# B&R Automation Studio project ACOPOStrakbyOk
Automation Studio 4.12.4.107 SP; technology packages: mappMotion 5.23.1

## Configuration Config1

CPU X20CP1586, AutomationRuntime E4.93, Build 4.1.2, Safety 0.0, Vc V4.72.6

### Task classes (Cpu.sw)
```
Cyclic#1 (cycle 800 us, tolerance 0 us):
  Vis <- Visualization.Vis.prg
Cyclic#4:
  StartMovem <- AssemblyControl.StartMovement.prg
DataObjects: McAcpSys
NcDataObjects: McDriveLog
Binaries: arsvcreg, udbdef, McAcpDrv, arflatprv, McProfGen, arcoal, FWRules, TCData, McAcpSim, ashwd, Config_1, ashwac, User, Config_4, sysconf, iomap, asfw, arconfig, Config_3, Config_2, Role
Libraries: McBase, McAxis, McAcpTrak, MpBase, operator, runtime, astime, AsIecCon, MpAxis, McAcpAx, AsBrStr, powerlnk, fileio, asepl, sys_lib
```

### Hardware
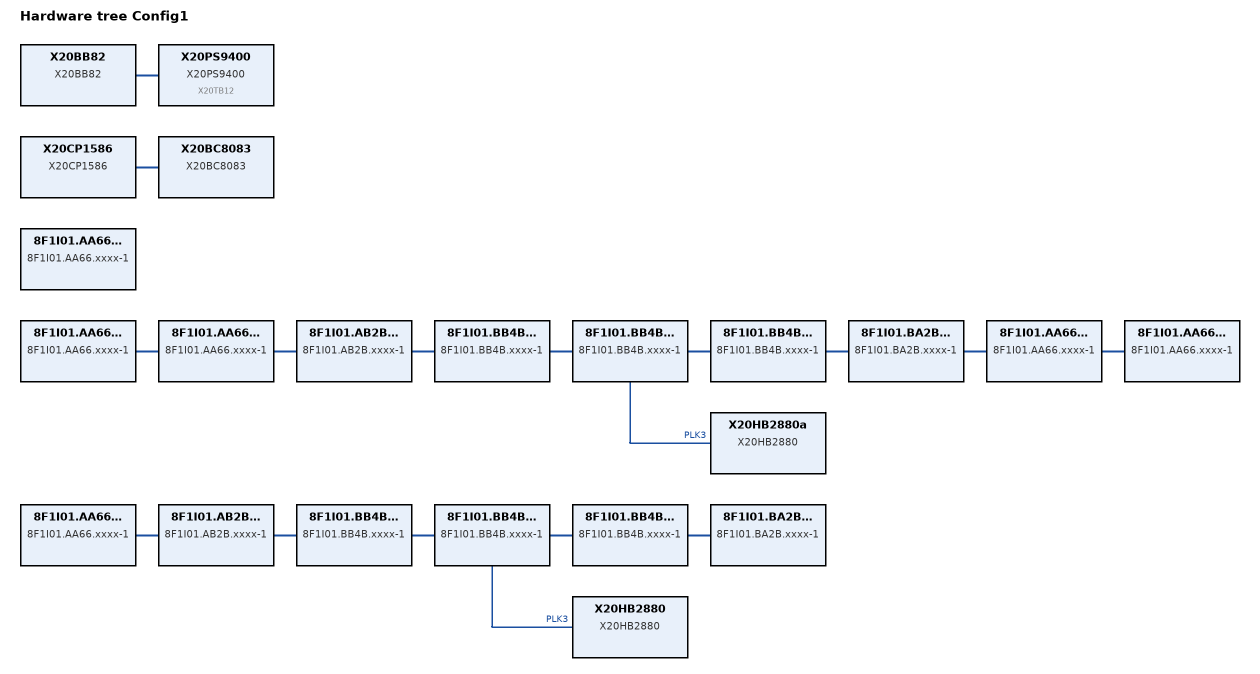
```
8F1I01.AA66.xxxx-1 : 8F1I01.AA66.xxxx-1 v1.0.0.2  [PLK1 -> 8F1I01.BA2B.xxxx-1a.PLK2 (NodeNumber=15) [Cable Type=PowerlinkCable, Length=10, Version=1.0.0.3]]
  DriveConfiguration:
    McTypeID = LLMConfig
  DriveConfiguration/Segment:
    Shape = STRAIGHT660
    SegmentReference = Seg_A_1
    SegmentSectorDirection = Positive
    ElongationCompensation = UseAssemblySetting
    StopReaction = UseAssemblySetting
    SpeedFilter = UseAssemblySetting
    PositionControllerLagMonitor = UseAssemblySetting
8F1I01.AA66.xxxx-1a : 8F1I01.AA66.xxxx-1 v1.0.0.2  [PLK2 -> 8F1I01.AA66.xxxx-1b.PLK1 (NodeNumber=14) [Cable Type=PowerlinkCable, Length=10, Version=1.0.0.3]]
  DriveConfiguration:
    McTypeID = LLMConfig
  DriveConfiguration/Segment:
    Shape = STRAIGHT660
    SegmentReference = Seg_A_2
    SegmentSectorDirection = Positive
    ElongationCompensation = UseAssemblySetting
    StopReaction = UseAssemblySetting
    SpeedFilter = UseAssemblySetting
    PositionControllerLagMonitor = UseAssemblySetting
8F1I01.AA66.xxxx-1b : 8F1I01.AA66.xxxx-1 v1.0.0.2  [PLK1 -> 8F1I01.AA66.xxxx-1a.PLK2 [Cable Type=PowerlinkCable, Length=10, Version=1.0.0.3]; PLK2 -> 8F1I01.AB2B.xxxx-1.PLK1 [Cable Type=PowerlinkCable, Length=10, Version=1.0.0.3]]
  DriveConfiguration:
    McTypeID = LLMConfig
  DriveConfiguration/Segment:
    Shape = STRAIGHT660
    SegmentReference = Seg_A_3
    SegmentSectorDirection = Positive
    ElongationCompensation = UseAssemblySetting
    StopReaction = UseAssemblySetting
    SpeedFilter = UseAssemblySetting
    PositionControllerLagMonitor = UseAssemblySetting
8F1I01.AA66.xxxx-1c : 8F1I01.AA66.xxxx-1 v1.0.0.2  [PLK1 -> 8F1I01.BA2B.xxxx-1.PLK2 [Cable Type=PowerlinkCable, Length=10, Version=1.0.0.3]; PLK2 -> 8F1I01.AA66.xxxx-1d.PLK1 [Cable Type=PowerlinkCable, Length=10, Version=1.0.0.3]]
  DriveConfiguration:
    McTypeID = LLMConfig
  DriveConfiguration/Segment:
    Shape = STRAIGHT660
    SegmentReference = Seg_A_9
    SegmentSectorDirection = Positive
    ElongationCompensation = UseAssemblySetting
    StopReaction = UseAssemblySetting
    SpeedFilter = UseAssemblySetting
    PositionControllerLagMonitor = UseAssemblySetting
8F1I01.AA66.xxxx-1d : 8F1I01.AA66.xxxx-1 v1.0.0.2  [PLK1 -> 8F1I01.AA66.xxxx-1c.PLK2 [Cable Type=PowerlinkCable, Length=10, Version=1.0.0.3]]
  DriveConfiguration:
    McTypeID = LLMConfig
  DriveConfiguration/Segment:
    Shape = STRAIGHT660
    SegmentReference = Seg_A_10
    SegmentSectorDirection = Positive
    ElongationCompensation = UseAssemblySetting
    StopReaction = UseAssemblySetting
    SpeedFilter = UseAssemblySetting
    PositionControllerLagMonitor = UseAssemblySetting
8F1I01.AA66.xxxx-1e : 8F1I01.AA66.xxxx-1 v1.0.0.2  [PLK2 -> 8F1I01.AB2B.xxxx-1a.PLK1 [Cable Type=PowerlinkCable, Length=10, Version=1.0.0.3]]
  DriveConfiguration:
    McTypeID = LLMConfig
  DriveConfiguration/Segment:
    Shape = STRAIGHT660
    SegmentReference = Seg_A_11
    SegmentSectorDirection = Positive
    ElongationCompensation = UseAssemblySetting
    StopReaction = UseAssemblySetting
    SpeedFilter = UseAssemblySetting
    PositionControllerLagMonitor = UseAssemblySetting
8F1I01.AB2B.xxxx-1 : 8F1I01.AB2B.xxxx-1 v1.0.0.2  [PLK1 -> 8F1I01.AA66.xxxx-1b.PLK2 [Cable Type=PowerlinkCable, Length=10, Version=1.0.0.3]; PLK2 -> 8F1I01.BB4B.xxxx-1.PLK1 [Cable Type=PowerlinkCable, Length=10, Version=1.0.0.3]]
  DriveConfiguration:
    McTypeID = LLMConfig
  DriveConfiguration/Segment:
    Shape = STRAIGHT105_TO_CIRCULAR
    SegmentReference = Seg_A_4
    SegmentSectorDirection = Positive
    ElongationCompensation = UseAssemblySetting
    StopReaction = UseAssemblySetting
    SpeedFilter = UseAssemblySetting
    PositionControllerLagMonitor = UseAssemblySetting
8F1I01.AB2B.xxxx-1a : 8F1I01.AB2B.xxxx-1 v1.0.0.2  [PLK1 -> 8F1I01.AA66.xxxx-1e.PLK2 [Cable Type=PowerlinkCable, Length=10, Version=1.0.0.3]; PLK2 -> 8F1I01.BB4B.xxxx-1c.PLK1 [Cable Type=PowerlinkCable, Length=10, Version=1.0.0.3]]
  DriveConfiguration:
    McTypeID = LLMConfig
  DriveConfiguration/Segment:
    Shape = STRAIGHT105_TO_CIRCULAR
    SegmentReference = Seg_A_12
    SegmentSectorDirection = Positive
    ElongationCompensation = UseAssemblySetting
    StopReaction = UseAssemblySetting
    SpeedFilter = UseAssemblySetting
    PositionControllerLagMonitor = UseAssemblySetting
8F1I01.BA2B.xxxx-1 : 8F1I01.BA2B.xxxx-1 v1.0.0.2  [PLK1 -> 8F1I01.BB4B.xxxx-1b.PLK2 [Cable Type=PowerlinkCable, Length=10, Version=1.0.0.3]; PLK2 -> 8F1I01.AA66.xxxx-1c.PLK1 [Cable Type=PowerlinkCable, Length=10, Version=1.0.0.3]]
  DriveConfiguration:
    McTypeID = LLMConfig
  DriveConfiguration/Segment:
    Shape = CIRCULAR_TO_STRAIGHT105
    SegmentReference = Seg_A_8
    SegmentSectorDirection = Positive
    ElongationCompensation = UseAssemblySetting
    StopReaction = UseAssemblySetting
    SpeedFilter = UseAssemblySetting
    PositionControllerLagMonitor = UseAssemblySetting
8F1I01.BA2B.xxxx-1a : 8F1I01.BA2B.xxxx-1 v1.0.0.2  [PLK1 -> 8F1I01.BB4B.xxxx-1e.PLK2 [Cable Type=PowerlinkCable, Length=10, Version=1.0.0.3]; PLK2 -> 8F1I01.AA66.xxxx-1.PLK1 [Cable Type=PowerlinkCable, Length=10, Version=1.0.0.3]]
  DriveConfiguration:
    McTypeID = LLMConfig
  DriveConfiguration/Segment:
    Shape = CIRCULAR_TO_STRAIGHT105
    SegmentReference = Seg_A_16
    SegmentSectorDirection = Positive
    ElongationCompensation = UseAssemblySetting
    StopReaction = UseAssemblySetting
    SpeedFilter = UseAssemblySetting
    PositionControllerLagMonitor = UseAssemblySetting
8F1I01.BB4B.xxxx-1 : 8F1I01.BB4B.xxxx-1 v1.0.0.2  [PLK1 -> 8F1I01.AB2B.xxxx-1.PLK2 [Cable Type=PowerlinkCable, Length=10, Version=1.0.0.3]; PLK2 -> 8F1I01.BB4B.xxxx-1a.PLK1 [Cable Type=PowerlinkCable, Length=10, Version=1.0.0.3]]
  DriveConfiguration:
    McTypeID = LLMConfig
  DriveConfiguration/Segment:
    Shape = CIRCULAR
    SegmentReference = Seg_A_5
    SegmentSectorDirection = Positive
    ElongationCompensation = UseAssemblySetting
    StopReaction = UseAssemblySetting
    SpeedFilter = UseAssemblySetting
    PositionControllerLagMonitor = UseAssemblySetting
8F1I01.BB4B.xxxx-1a : 8F1I01.BB4B.xxxx-1 v1.0.0.2  [PLK1 -> 8F1I01.BB4B.xxxx-1.PLK2 (NodeNumber=8) [Cable Type=PowerlinkCable, Length=10, Version=1.0.0.3]; PLK2 -> 8F1I01.BB4B.xxxx-1b.PLK1 (NodeNumber=8) [Cable Type=PowerlinkCable, Length=10, Version=1.0.0.3]; PLK3 -> X20HB2880a.ETH1 (NodeNumber=8) [Cable Type=PowerlinkCable, Length=10, Version=1.0.0.3]]
  DriveConfiguration:
    McTypeID = LLMConfig
  DriveConfiguration/Segment:
    Shape = CIRCULAR
    SegmentReference = Seg_A_6
    SegmentSectorDirection = Positive
    ElongationCompensation = UseAssemblySetting
    StopReaction = UseAssemblySetting
    SpeedFilter = UseAssemblySetting
    PositionControllerLagMonitor = UseAssemblySetting
8F1I01.BB4B.xxxx-1b : 8F1I01.BB4B.xxxx-1 v1.0.0.2  [PLK1 -> 8F1I01.BB4B.xxxx-1a.PLK2 [Cable Type=PowerlinkCable, Length=10, Version=1.0.0.3]; PLK2 -> 8F1I01.BA2B.xxxx-1.PLK1 [Cable Type=PowerlinkCable, Length=10, Version=1.0.0.3]]
  DriveConfiguration:
    McTypeID = LLMConfig
  DriveConfiguration/Segment:
    Shape = CIRCULAR
    SegmentReference = Seg_A_7
    SegmentSectorDirection = Positive
    ElongationCompensation = UseAssemblySetting
    StopReaction = UseAssemblySetting
    SpeedFilter = UseAssemblySetting
    PositionControllerLagMonitor = UseAssemblySetting
8F1I01.BB4B.xxxx-1c : 8F1I01.BB4B.xxxx-1 v1.0.0.2  [PLK1 -> 8F1I01.AB2B.xxxx-1a.PLK2 [Cable Type=PowerlinkCable, Length=10, Version=1.0.0.3]; PLK2 -> 8F1I01.BB4B.xxxx-1d.PLK1 [Cable Type=PowerlinkCable, Length=10, Version=1.0.0.3]]
  DriveConfiguration:
    McTypeID = LLMConfig
  DriveConfiguration/Segment:
    Shape = CIRCULAR
    SegmentReference = Seg_A_13
    SegmentSectorDirection = Positive
    ElongationCompensation = UseAssemblySetting
    StopReaction = UseAssemblySetting
    SpeedFilter = UseAssemblySetting
    PositionControllerLagMonitor = UseAssemblySetting
8F1I01.BB4B.xxxx-1d : 8F1I01.BB4B.xxxx-1 v1.0.0.2  [PLK1 -> 8F1I01.BB4B.xxxx-1c.PLK2 (NodeNumber=2) [Cable Type=PowerlinkCable, Length=10, Version=1.0.0.3]; PLK2 -> 8F1I01.BB4B.xxxx-1e.PLK1 (NodeNumber=2) [Cable Type=PowerlinkCable, Length=10, Version=1.0.0.3]; PLK3 -> X20HB2880.ETH1 (NodeNumber=2) [Cable Type=PowerlinkCable, Length=10, Version=1.0.0.3]]
  DriveConfiguration:
    McTypeID = LLMConfig
  DriveConfiguration/Segment:
    Shape = CIRCULAR
    SegmentReference = Seg_A_14
    SegmentSectorDirection = Positive
    ElongationCompensation = UseAssemblySetting
    StopReaction = UseAssemblySetting
    SpeedFilter = UseAssemblySetting
    PositionControllerLagMonitor = UseAssemblySetting
8F1I01.BB4B.xxxx-1e : 8F1I01.BB4B.xxxx-1 v1.0.0.2  [PLK1 -> 8F1I01.BB4B.xxxx-1d.PLK2 [Cable Type=PowerlinkCable, Length=10, Version=1.0.0.3]; PLK2 -> 8F1I01.BA2B.xxxx-1a.PLK1 [Cable Type=PowerlinkCable, Length=10, Version=1.0.0.3]]
  DriveConfiguration:
    McTypeID = LLMConfig
  DriveConfiguration/Segment:
    Shape = CIRCULAR
    SegmentReference = Seg_A_15
    SegmentSectorDirection = Positive
    ElongationCompensation = UseAssemblySetting
    StopReaction = UseAssemblySetting
    SpeedFilter = UseAssemblySetting
    PositionControllerLagMonitor = UseAssemblySetting
X20BB82 : X20BB82 v1.1.0.0
X20BC8083 : X20BC8083 v2.14.0.0  [PLK1 -> X20CP1586.IF3 (NodeNumber=1) [Cable Type=PowerlinkCable, Length=10, Version=1.0.0.3]; SL -> X20BB82.SL1]
X20CP1586 : X20CP1586 v1.10.0.0
  Connector IF2:
    ActivateDevice = 1
  Connector IF3:
    CycleTime = 800
  ConfigurationID = ACOPOStrakbyOk_Config1
  Simulation = 1
  MotionLoggerSize = 2048000
  TimerDeviceType = EPLX2X
  TimerDevice = X20CP1586.IF3
  TaskClassIdleTime = 1600
  Cyclic1Duration = 800
  Cyclic1Tolerance = 0
  Cyclic3Duration = 49600
  Cyclic3Tolerance = 49600
  Cyclic8Duration = 9600
  FileDevice1
  FileDeviceName1 = SvgData
  FileDevicePath1 = C:\projects\TestACO\ACOPOStrakbyOk\SvgData
X20HB2880 : X20HB2880 v1.2.0.0  [ETH1 -> 8F1I01.BB4B.xxxx-1d.PLK3 [Cable Type=PowerlinkCable, Length=10, Version=1.0.0.3]; SS -> X20BB82.SS2]
X20HB2880a : X20HB2880 v1.2.0.0  [ETH1 -> 8F1I01.BB4B.xxxx-1a.PLK3 [Cable Type=PowerlinkCable, Length=10, Version=1.0.0.3]; SS -> X20BB82.SS1]
X20PS9400 : X20PS9400 v1.8.0.0  [SS1 -> X20TB12a.SS; PS -> X20BB82.PS1]
X20TB12a : X20TB12 v1.0.0.0
```

### Config_1.assembly - X20CP1586/mappMotion/TrakOval/Config_1.assembly
```
Element gAssembly_1 (Type=assembly)
  Tracks:
    TrackSeparation = 0.030
    Track[1]:
      Segments:
        SegmentRef[1] = ::Seg_A_1
        SegmentRef[2] = ::Seg_A_2
        SegmentRef[3] = ::Seg_A_3
        SegmentRef[4] = ::Seg_A_4
        SegmentRef[5] = ::Seg_A_5
        SegmentRef[6] = ::Seg_A_6
        SegmentRef[7] = ::Seg_A_7
        SegmentRef[8] = ::Seg_A_8
        SegmentRef[9] = ::Seg_A_9
        SegmentRef[10] = ::Seg_A_10
        SegmentRef[11] = ::Seg_A_11
        SegmentRef[12] = ::Seg_A_12
        SegmentRef[13] = ::Seg_A_13
        SegmentRef[14] = ::Seg_A_14
        SegmentRef[15] = ::Seg_A_15
        SegmentRef[16] = ::Seg_A_16
      Position = Absolute
        SegmentRef = ::Seg_A_1
        SegmentCountDirection = RightToLeft
        Translation:
          X = 0.0
          Y = 0.0
          Z = 0.0
        Orientation:
          Angle1 = 0.0
          Angle2 = 0.0
          Angle3 = 180
  CommonSegmentSettings:
    SegmentSimulationOnPLC = Off
    CoggingCompensation = Active
      UpperVelLimit = 0.5
    ElongationCompensation = Inactive
    StopReaction = InductionHalt
    SpeedFilter = NotUsed
    ControllerParameters:
      DefaultParameter:
        Controller:
          Position:
            ProportionalGain = 200
          Speed:
            ProportionalGain = 80
            IntegrationTime = 0.0
          FeedForward:
            TotalMass = 1
            ForcePositive = 0.0
            ForceNegative = 0.0
            SpeedForceFactor = 0.0
            ForceLoad = 0.0
        MovementErrorLimits:
          PositionError = 0.001
          VelocityError = 0.05
        Diverter:
          ForceOverride = 1.0
      AdditionalParameterSets = NotUsed
    ScopeOfErrorReaction = Assembly
    ShuttleIdentificationTime = 0
    PositionControllerLagMonitor = Inactive
    Diverter:
      DiverterWeakEndOverrideFactor = 1.0
      DiverterStrenEndOverrideFactor = 1.0
  Shuttles:
    MaxShuttleCount = 25
    MaxShuttleCommandCount = 0
    Deceleration = 0.0
    UseConvoys = Inactive
    DistanceReserve:
      Collision = 0.002
      ErrorStop = 0.006
    ShuttleStereotypes:
      ShuttleStRef[1] = ShuttleStereotype_1
    MagnetPlateConfigurations:
      ShuttleType[1] = 8F1SA.100.xxxxxx-x
    CollisionAvoidance:
      Strategy = Constant
      Exclusion = NotUsed
      MaximumModelDimensions:
        Length:
          ExtentToFront = 0.05
          ExtentToBack = 0.05
        Width:
          Width = 0.040
    Coupling:
      CouplingFeature:
        EliminateShuttleToShuttleDelay = FALSE
  AssemblyFeatures:
    AssemblyFeatureRef[1] = Feature_Sim_Shuttle_Def_1
  Visualization:
    MonitoringPv = gShuttleMon
    ProcessingTaskClass = 1
  Alarms = None
```

### Config_2.shuttlestereotype - X20CP1586/mappMotion/TrakOval/Config_2.shuttlestereotype
```
Element ShuttleStereotype_1 (Type=shuttlestereotype)
  MeasurementUnit = 5067858
  MeasurementResolution = 0.00001
  MovementLimits = Internal
    VelocityIsReadOnly = 0
    Velocity:
      Velocity = 4
    AccelerationIsReadOnly = 0
    Acceleration:
      Acceleration = 40
    DecelerationIsReadOnly = 0
    Deceleration:
      Deceleration = 40
    UpdateMode = Immediately
  JerkFilter = NotUsed
  UserData:
    Size = 12
  StateTransitions:
    AutomaticRecontrol = Active
```

### Config_4.assemblyfeature - X20CP1586/mappMotion/TrakOval/Config_4.assemblyfeature
```
Element Feature_Sim_Shuttle_Def_1 (Type=assemblyfeature)
  Type = InitShuttleSim
    InitShuttleSim[1]:
      SectorRef = SectorTrackA
      Orientation = Positive
      ShuttleDefinition = ShuttleSetDefinition
        StartPosition = 0.3
        NumberOfShuttles = 5
        DistnaceBetweenShuttles = 0.2
```

## Logical view

Binary libraries used (declarations not repeated): operator, runtime, astime, AsIecCon, McBase, McAxis, McAcpTrak 5.23.1, MpBase, MpAxis, McAcpAx, AsBrStr

### Global.typ - Global data types
```iecst
(* Shuttle user data structure *)
TYPE
    ShuttleUserData_type : STRUCT
        Color : ShuttleColor_enum; (* Example: product colour *)
        Weight : REAL; (* Example: product weight *)
        PartNumber : UDINT; (* Example: product part number *)
    END_STRUCT;

    ShuttleColor_enum :
    (
        ORANGE,
        GREEN,
        RED,
        BLUE,
        WHITE
    );
END_TYPE

(* Assembly interface *)
TYPE
    TrakAsmCommand_type : STRUCT
        Power : BOOL;
        ShuttleStart : BOOL;
        ShuttleStop : BOOL;
        Reset : BOOL;
    END_STRUCT;

    TrakAsmParameter_type : STRUCT
        Velocity : REAL;
        Acceleration : REAL;
        Deceleration : REAL;
    END_STRUCT;

    TrakAsmStatus_type : STRUCT
        Disabled : BOOL;
        Ready : BOOL;
        Homing : BOOL;
        Stopping : BOOL;
        ErrorStop : BOOL;
    END_STRUCT;

    TrakAsm_type : STRUCT
        Command : TrakAsmCommand_type;
        Parameter : TrakAsmParameter_type;
        Status : TrakAsmStatus_type;
        ShuttleCnt : UINT;
    END_STRUCT;
END_TYPE
```

### Global.var - Global variables
```iecst
(* Assembly interface *)
VAR
    gTrakAsm : TrakAsm_type;
END_VAR

(* Shuttle user data structure *)
VAR
    gShuttleUserData : ShuttleUserData_type;
END_VAR

(* Shuttle monitor structure for Vis *)
VAR
    gShuttleMon : McAcpTrakAssemblyMonData;
END_VAR
```


### Program Logical/AssemblyControl/StartMovement

#### Variables.var
```iecst
(* Constants *)
VAR CONSTANT
    MAX_SHUTTLE_CNT : USINT := 25; (* Maximum number of shuttles handled by the assembly *)
END_VAR

(* Sequence control *)
VAR
    Step : StepEnum;
    CurrentShuttleNumber : UINT;
    ShuttleReferences : ARRAY[1..MAX_SHUTTLE_CNT] OF McAxisType;
    UserDataSize : UDINT;
END_VAR

(* Function blocks *)
VAR
    MC_BR_AsmPowerOn_AcpTrak_0 : MC_BR_AsmPowerOn_AcpTrak;
    MC_BR_AsmPowerOff_AcpTrak_0 : MC_BR_AsmPowerOff_AcpTrak;
    MC_BR_AsmGetShuttle_AcpTrak_0 : MC_BR_AsmGetShuttle_AcpTrak;
    MC_BR_AsmStop_AcpTrak_0 : MC_BR_AsmStop_AcpTrak;
    MC_BR_AsmReadStatus_AcpTrak_0 : MC_BR_AsmReadStatus_AcpTrak;
    MC_BR_AsmReset_AcpTrak_0 : MC_BR_AsmReset_AcpTrak;
    MC_BR_RoutedMoveVel_AcpTrak_0 : MC_BR_RoutedMoveVel_AcpTrak;
END_VAR
```

#### Main.st
```iecst
PROGRAM _INIT
    (* Initialize parameters for shuttle movements. *)
    gTrakAsm.Parameter.Velocity := 2.0;
    gTrakAsm.Parameter.Acceleration := 20.0;
    gTrakAsm.Parameter.Deceleration := 20.0;

    (* Write this value into the size of user data in the shuttle stereotype configuration. *)
    UserDataSize := SIZEOF(gShuttleUserData);

    (* Set the assembly reference for all assembly function blocks. *)
    MC_BR_AsmPowerOn_AcpTrak_0.Assembly     := ADR(gAssembly_1);
    MC_BR_AsmPowerOff_AcpTrak_0.Assembly    := ADR(gAssembly_1);
    MC_BR_AsmStop_AcpTrak_0.Assembly        := ADR(gAssembly_1);
    MC_BR_AsmGetShuttle_AcpTrak_0.Assembly  := ADR(gAssembly_1);
    MC_BR_AsmReadStatus_AcpTrak_0.Assembly  := ADR(gAssembly_1);
    MC_BR_AsmReset_AcpTrak_0.Assembly       := ADR(gAssembly_1);

    (* Enable reading of current status of the assembly. *)
    MC_BR_AsmReadStatus_AcpTrak_0.Enable := TRUE;

    (* Initialize constant parameters for routed moves. *)
    MC_BR_RoutedMoveVel_AcpTrak_0.Sector        := ADR(SectorTrackA);
    MC_BR_RoutedMoveVel_AcpTrak_0.Jerk          := 0.0;
    MC_BR_RoutedMoveVel_AcpTrak_0.BufferMode    := mcABORTING;
    MC_BR_RoutedMoveVel_AcpTrak_0.AdvancedParameters.StartDirection     := mcDIR_UNDEFINED;
    MC_BR_RoutedMoveVel_AcpTrak_0.AdvancedParameters.EndDirection       := mcDIR_POSITIVE;
    MC_BR_RoutedMoveVel_AcpTrak_0.AdvancedParameters.ShuttleOrientation := mcDIR_UNDEFINED;

    (* Initialize constant parameter for assembly stop command. *)
    MC_BR_AsmStop_AcpTrak_0.StopMode := mcSTOPMODE_JERK_LIMIT;
END_PROGRAM

PROGRAM _CYCLIC
    IF gTrakAsm.Status.ErrorStop THEN
        Step := ERROR;
    END_IF

    CASE Step OF

        (* Power off assembly and wait for power on command *)
        POWER_OFF:
            (* Assembly is already powered off. *)
            IF gTrakAsm.Status.Disabled THEN
                Step := POWERED_OFF;
            ELSE
                MC_BR_AsmPowerOff_AcpTrak_0.Execute := TRUE;
                Step := WAIT_POWER_OFF;
            END_IF

        (* The assembly is being powered off. *)
        WAIT_POWER_OFF:
            (* Power off is done. *)
            IF MC_BR_AsmPowerOff_AcpTrak_0.Done THEN
                MC_BR_AsmPowerOff_AcpTrak_0.Execute := FALSE;
                Step := POWERED_OFF;
            ELSIF MC_BR_AsmPowerOff_AcpTrak_0.Error THEN
                Step := ERROR;
            END_IF

        (* The assembly is powered off, wait for a command to power it on. *)
        POWERED_OFF:
            (* The assembly is to be powered on. *)
            IF gTrakAsm.Command.Power THEN
                Step := POWER_ON;
            END_IF

        (* Power on assembly *)
        POWER_ON:
            MC_BR_AsmPowerOn_AcpTrak_0.Execute := TRUE;
            Step := WAIT_POWER_ON;

        (* The assembly is being powered on. *)
        WAIT_POWER_ON:
            (* Assembly is not yet powered on. *)
            IF MC_BR_AsmPowerOn_AcpTrak_0.Done THEN
                MC_BR_AsmPowerOn_AcpTrak_0.Execute := FALSE;

                (* Store the shuttles in the shuttle array. On real hardware, the set of shuttles might have changed. *)
                CurrentShuttleNumber := 1;
                brsmemset(ADR(ShuttleReferences), 0, SIZEOF(ShuttleReferences));
                Step := GET_SHUTTLE;
            ELSIF MC_BR_AsmPowerOn_AcpTrak_0.Error THEN
                Step := ERROR;
            END_IF

        (* Get all shuttles on the assembly (those physically available on the real hardware or the added ones in the simulation, resp.). *)
        GET_SHUTTLE:
            MC_BR_AsmGetShuttle_AcpTrak_0.Enable := TRUE;

            IF MC_BR_AsmGetShuttle_AcpTrak_0.Valid THEN
                (* There are no shuttles on the assembly. *)
                IF MC_BR_AsmGetShuttle_AcpTrak_0.TotalCount = 0 THEN
                    gTrakAsm.ShuttleCnt := 0;
                    MC_BR_AsmGetShuttle_AcpTrak_0.Enable := FALSE;
                    MC_BR_AsmGetShuttle_AcpTrak_0.Next := FALSE;

                    Step := READY;
                (* As soon as the next shuttle has been output by the function block, RemainingCount
                   is reduced and this condition becomes true. *)
                ELSIF (MC_BR_AsmGetShuttle_AcpTrak_0.RemainingCount <> (MC_BR_AsmGetShuttle_AcpTrak_0.TotalCount - CurrentShuttleNumber)) THEN
                    CurrentShuttleNumber := CurrentShuttleNumber + 1;
                    MC_BR_AsmGetShuttle_AcpTrak_0.Next := FALSE;
                ELSE
                    (* Store all axis references in an array for global movement commands. *)
                    ShuttleReferences[CurrentShuttleNumber] := MC_BR_AsmGetShuttle_AcpTrak_0.Axis;
                    (* Get next shuttle reference with positive edge on .Next. *)
                    MC_BR_AsmGetShuttle_AcpTrak_0.Next := TRUE;

                    (* All shuttles have been stored. *)
                    IF (MC_BR_AsmGetShuttle_AcpTrak_0.RemainingCount = 0) THEN
                        gTrakAsm.ShuttleCnt := MC_BR_AsmGetShuttle_AcpTrak_0.TotalCount;
                        MC_BR_AsmGetShuttle_AcpTrak_0.Enable := FALSE;
                        MC_BR_AsmGetShuttle_AcpTrak_0.Next := FALSE;

                        Step := READY;
                    END_IF
                END_IF
            END_IF

        (* Assembly is active and ready for movement. *)
        READY:
            (* Power off the assembly. *)
            IF NOT gTrakAsm.Command.Power THEN
                Step := POWER_OFF;
            (* Wait for movement command if shuttles are present. *)
            ELSIF gTrakAsm.Command.ShuttleStart AND gTrakAsm.ShuttleCnt > 0 THEN
                gTrakAsm.Command.ShuttleStart := FALSE;
                CurrentShuttleNumber := 1;
                Step := START_MOVEMENT;
            END_IF

        (* Move all shuttles on assembly to the same target position with the same velocity. *)
        (* Used for startup to accelerate all shuttles to an initial velocity in order to
           pass the first process-point. *)
        START_MOVEMENT:
            IF CurrentShuttleNumber <= gTrakAsm.ShuttleCnt THEN
                MC_BR_RoutedMoveVel_AcpTrak_0.Axis          := ADR(ShuttleReferences[CurrentShuttleNumber]);
                MC_BR_RoutedMoveVel_AcpTrak_0.Position      := 0.3 + gTrakAsm.ShuttleCnt * 0.15;
                MC_BR_RoutedMoveVel_AcpTrak_0.Velocity      := gTrakAsm.Parameter.Velocity;
                MC_BR_RoutedMoveVel_AcpTrak_0.RouteVelocity := gTrakAsm.Parameter.Velocity;
                MC_BR_RoutedMoveVel_AcpTrak_0.Acceleration  := gTrakAsm.Parameter.Acceleration;
                MC_BR_RoutedMoveVel_AcpTrak_0.Deceleration  := gTrakAsm.Parameter.Deceleration;
                MC_BR_RoutedMoveVel_AcpTrak_0.Execute       := TRUE;

                Step := WAIT_START_MOVEMENT;
            ELSE
                Step := MOVING;
            END_IF

        (* Wait until a shuttle movement is active. *)
        WAIT_START_MOVEMENT:
            IF MC_BR_RoutedMoveVel_AcpTrak_0.Active THEN
                MC_BR_RoutedMoveVel_AcpTrak_0.Execute := FALSE;
                CurrentShuttleNumber := CurrentShuttleNumber + 1;
                Step := START_MOVEMENT;
            (* There is invalid speed or acceleration setting or shuttle caused an error stop. *)
            ELSIF MC_BR_RoutedMoveVel_AcpTrak_0.Error THEN
                Step := ERROR;
            END_IF

        (* A movement has been started for all shuttles. *)
        MOVING:
            (* Wait for Stop command. *)
            IF gTrakAsm.Command.ShuttleStop THEN
                gTrakAsm.Command.ShuttleStop := FALSE;
                Step := STOPPING;
            END_IF

        (* Stop all shuttles with specified deceleration at their current locations. *)
        STOPPING:
            MC_BR_AsmStop_AcpTrak_0.Execute := TRUE;
            Step := WAIT_STOPPING;

        (* Wait until all shuttles are stopped. *)
        WAIT_STOPPING:
            IF MC_BR_AsmStop_AcpTrak_0.Done THEN
                MC_BR_AsmStop_AcpTrak_0.Execute := FALSE;
                Step := READY;
            (* A shuttle caused an error stop. *)
            ELSIF MC_BR_AsmStop_AcpTrak_0.Error THEN
                Step := ERROR;
            END_IF

        (* An error occured on the assembly. *)
        ERROR:
            (* Wait for the user to trigger the error reset. *)
            IF gTrakAsm.Command.Reset THEN
                gTrakAsm.Command.Reset := FALSE;
                MC_BR_AsmReset_AcpTrak_0.Execute := TRUE;
                Step := RESET;
            END_IF

        (* Reset assembly due to an error. *)
        RESET:
            IF MC_BR_AsmReset_AcpTrak_0.Done THEN
                gTrakAsm.Command.ShuttleStart           := FALSE;
                gTrakAsm.Command.ShuttleStop            := FALSE;
                MC_BR_AsmReset_AcpTrak_0.Execute        := FALSE;
                MC_BR_AsmPowerOn_AcpTrak_0.Execute      := FALSE;
                MC_BR_AsmPowerOff_AcpTrak_0.Execute     := FALSE;
                MC_BR_AsmStop_AcpTrak_0.Execute         := FALSE;
                MC_BR_RoutedMoveVel_AcpTrak_0.Execute   := FALSE;

                Step := READY;
            END_IF
    END_CASE

    (* Read assembly status cyclically to assembly interface. *)
    gTrakAsm.Status.Disabled  := MC_BR_AsmReadStatus_AcpTrak_0.AssemblyDisabled;
    gTrakAsm.Status.Ready     := MC_BR_AsmReadStatus_AcpTrak_0.AssemblyReady;
    gTrakAsm.Status.Homing    := MC_BR_AsmReadStatus_AcpTrak_0.AssemblyHoming;
    gTrakAsm.Status.Stopping  := MC_BR_AsmReadStatus_AcpTrak_0.AssemblyStopping;
    gTrakAsm.Status.ErrorStop := MC_BR_AsmReadStatus_AcpTrak_0.AssemblyErrorStop;

    (* Cyclic function blocks calls *)
    MC_BR_AsmPowerOn_AcpTrak_0();
    MC_BR_AsmGetShuttle_AcpTrak_0();
    MC_BR_AsmPowerOff_AcpTrak_0();
    MC_BR_AsmStop_AcpTrak_0();
    MC_BR_RoutedMoveVel_AcpTrak_0();
    MC_BR_AsmReadStatus_AcpTrak_0();
    MC_BR_AsmReset_AcpTrak_0();
END_PROGRAM
```

- Visualisation Logical/Visualization (not shown)
